(* IEC 61131-3 sources: T4Exjobb/Sigma/Stations/MachineControl/MachineControl/Class/TCPv2, 1 file *)

(* ---- TCPv2.st ---- *)
(*!
<Class
	Name               = "TCPv2"
	Revision           = "0.0"
	RealtimeTask       = "false"
	CyclicTask         = "true"
	BackgroundTask     = "false"
	Sigmatek           = "false"
	OSInterface        = "false"
	HighPriority       = "false"
	Automatic          = "false"
	UpdateMode         = "Prescan"
	SharedCommandTable = "true"
	Objectsize         = "(376,120)">
	<Channels>
		<Server Name="ClassSvr" Visualized="false" Initialize="false" WriteProtected="true" Retentive="false"/>
		<Server Name="goOnline" Visualized="false" Initialize="false" WriteProtected="false" Retentive="false"/>
		<Server Name="isOnline" Visualized="false" Initialize="false" WriteProtected="true" Retentive="false"/>
		<Server Name="SendReturn" Visualized="false" Initialize="false" WriteProtected="true" Retentive="false"/>
		<Client Name="Client" Required="true" Internal="true"/>
		<Client Name="cPort" Required="true" Internal="false" Comment="port number ... must be connected or initialized"/>
		<Client Name="ocIP" Required="true" Internal="false"/>
	</Channels>
	<Network Name="TCPv2">
		<!-- List of Components in this network -->
		<Components>
			<Object
				Name           = "Client"
				Class          = "_TCPIP_CLIENT"
				Position       = "(240,120)"
				Visualized     = "true"
				Remotely       = "true"
				CyclicTime     = "10 ms"
				BackgroundTime = "always">
				<Channels>
					<Server Name="Control"/>
					<Server Name="SemaName01"/>
					<Server Name="SemaName02"/>
					<Server Name="TaskName"/>
					<Client Name="cConfig"/>
					<Client Name="cMaxConnections" Value="1"/>
					<Client Name="co_MultiTask"/>
					<Client Name="co_SigCLib"/>
					<Client Name="co_StdLib"/>
					<Client Name="co_Task"/>
					<Client Name="cPort" Value="502"/>
					<Client Name="cSizeOfTXBuffer"/>
				</Channels>
			</Object>
		</Components>
		<Comments>
		</Comments>
		<!-- List of Connections in this network -->
		<Connections>
			<Connection Source="this.Client" Destination="Client.Control"/>
			<Connection Source="Client.cPort" Destination="this.cPort" Vertices="(240,210),(38,210),"/>
		</Connections>
		<!-- Headerfiles -->
		<Options>
		</Options>
	</Network>
</Class>
*)
TCPv2 : CLASS
  //Servers:
	ClassSvr 	: SvrChCmd_DINT;
	goOnline 	: SvrCh_DINT;
	isOnline 	: SvrCh_DINT;
	SendReturn 	: SvrCh_DINT;
  //Clients:
	cPort 	: CltCh_DINT;
	Client 	: CltChCmd__TCPIP_CLIENT;
	ocIP 	: CltChCmd_String;
  //Variables:
		handle 	: DINT;
		IPaddr : ARRAY [0..20] OF CHAR;

  //Functions:

	FUNCTION VIRTUAL GLOBAL Init;

	FUNCTION VIRTUAL GLOBAL CyWork
		VAR_INPUT
			EAX 	: UDINT;
		END_VAR
		VAR_OUTPUT
			state (EAX) 	: UDINT;
		END_VAR;

	FUNCTION GLOBAL Send
		VAR_INPUT
			pData 	: ^void;
			udSize 	: UDINT;
		END_VAR
		VAR_OUTPUT
			retcode 	: DINT;
		END_VAR;

	FUNCTION VIRTUAL DataCallback
		VAR_INPUT
			pData 	: ^void;
			udSize 	: UDINT;
		END_VAR;

	FUNCTION VIRTUAL GLOBAL goOnline::Write
		VAR_INPUT
			input (EAX) 	: DINT;
		END_VAR
		VAR_OUTPUT
			result (EAX) 	: DINT;
		END_VAR;
  //Tables:
	FUNCTION @STD
		VAR_OUTPUT
			ret_code	: CONFSTATES;
		END_VAR;
	FUNCTION GLOBAL TAB @CT_;
END_CLASS;

#pragma using _TCPIP_CLIENT
#pragma usingLtd String

FUNCTION VIRTUAL TCPv2::DataCallback
	VAR_INPUT
		pData 	: ^void;
		udSize 	: UDINT;
	END_VAR

  TRACE("CALLBACK");

END_FUNCTION

FUNCTION VIRTUAL GLOBAL TCPv2::CyWork
	VAR_INPUT
		EAX 	: UDINT;
	END_VAR
	VAR_OUTPUT
		state (EAX) 	: UDINT;
	END_VAR

  isOnline := Client.IsConnected(dHandle:=handle);

	state := READY;

END_FUNCTION

FUNCTION GLOBAL TCPv2::Send
	VAR_INPUT
		pData 	: ^void;
		udSize 	: UDINT;
	END_VAR
	VAR_OUTPUT
		retcode 	: DINT;
	END_VAR

  retcode := Client.SendData(pData:=pData, udSize:=udSize, dHandle:=handle, bDirect:=0);

END_FUNCTION

FUNCTION VIRTUAL GLOBAL TCPv2::goOnline::Write
	VAR_INPUT
		input (EAX) 	: DINT;
	END_VAR
	VAR_OUTPUT
		result (EAX) 	: DINT;
	END_VAR

	goOnline := input;

  if goOnline = 1 then
    handle := Client.AddConnection(pIPAddress:=#IPaddr[0], pCallbackThis:=this, pCallbackMeth:=#DataCallback(), udTimeout:=100);
  else
    Client.DelConnection(dHandle:=handle);
  end_if;

	result := goOnline;

END_FUNCTION

FUNCTION VIRTUAL GLOBAL TCPv2::Init

  if _FirstScan then
    ocIP.ReadDataOff(udOff:=0, pData:=#IPaddr[0], udMax:=ocIP.GetLength());
  end_if;

END_FUNCTION
